// TIA Portal V17 program export: 0 tag tables, 1 data types, 3 data blocks, 1 code blocks (in call order from the OBs), 4 instance data blocks

TYPE "sPut"
// stored: IsFailsafeCompliant false
   STRUCT
      tP : Struct
         REQ : Bool;   // OUT Start sending data
         ERROR : Bool;   // OUT Error sending data
         DONE : Bool;   // OUT sending data completed successfully
         status : Int;
      END_STRUCT;
   END_STRUCT;
END_TYPE

DATA_BLOCK "Data_send_1"   // DB1
{ S7_Optimized_Access := 'FALSE' }
VERSION : 0.1
// stored: AutoNumber true, IsOnlyStoredInLoadMemory false, IsWriteProtectedInAS false
   VAR
      Bool_1 : Bool;
      Bool_2 : Bool;
      Bool_3 : Bool;
      Bool_4 : Bool;
   END_VAR
BEGIN
END_DATA_BLOCK

DATA_BLOCK "dbReceive_PLC1fromPLC2"   // DB7
{ S7_Optimized_Access := 'TRUE' }
VERSION : 0.1
// stored: AutoNumber true, IsOnlyStoredInLoadMemory false, IsWriteProtectedInAS false
   VAR
      Odebrane : Int;
   END_VAR
BEGIN
END_DATA_BLOCK

DATA_BLOCK "dbSend_PLC1toPLC2"   // DB4
{ S7_Optimized_Access := 'TRUE' }
VERSION : 0.1
// stored: AutoNumber true, IsOnlyStoredInLoadMemory false, IsWriteProtectedInAS false
   VAR
      wyslane : Int;
   END_VAR
BEGIN
END_DATA_BLOCK

ORGANIZATION_BLOCK "Main"   // OB1, LAD, ProgramCycle
TITLE = "Main Program Sweep (Cycle)"
{ S7_Optimized_Access := 'TRUE' }
VERSION : 0.1
// stored: AutoNumber true, IsIECCheckEnabled false, SetENOAutomatically false
BEGIN
END_ORGANIZATION_BLOCK

DATA_BLOCK "IEC_Counter_0_DB"   // DB5
{ S7_Optimized_Access := 'TRUE' }
// stored: AutoNumber true, InstanceOfName IEC_COUNTER, OfSystemLibElement IEC_COUNTER, OfSystemLibVersion 1.0
"IEC_COUNTER"
   // VAR RETAIN
   //    CU : Bool;
   //    CD : Bool;
   //    R : Bool;
   //    LD : Bool;
   //    QU : Bool;
   //    QD : Bool;
   //    PV : Int;
   //    CV : Int;
   // END_VAR
BEGIN
END_DATA_BLOCK

DATA_BLOCK "PUT_DB"   // DB2
// stored: AutoNumber true, InstanceOfName PUT_SFB, OfSystemLibElement PUT, OfSystemLibVersion 1.3
"PUT_SFB"
   // VAR_INPUT
   //    REQ : Bool;
   //    ID : Word;
   // END_VAR
   // VAR_OUTPUT
   //    DONE : Bool;
   //    ERROR : Bool;
   //    STATUS : Word;
   // END_VAR
   // VAR_IN_OUT
   //    ADDR_1 : Remote;
   //    ADDR_2 : Remote;
   //    ADDR_3 : Remote;
   //    ADDR_4 : Remote;
   //    SD_1 : Variant;
   //    SD_2 : Variant;
   //    SD_3 : Variant;
   //    SD_4 : Variant;
   // END_VAR
BEGIN
END_DATA_BLOCK

DATA_BLOCK "TRCV_C_DB_1"   // DB6
// stored: AutoNumber true, InstanceOfName TRCV_C, OfSystemLibElement TRCV_C, OfSystemLibVersion 2.1
"TRCV_C"
   // VAR_INPUT
   //    EN_R : Bool;
   //    CONT : Bool;
   //    LEN : UInt;
   // END_VAR
   // VAR_OUTPUT
   //    DONE : Bool;
   //    BUSY : Bool;
   //    ERROR : Bool;
   //    STATUS : Word;
   //    RCVD_LEN : UInt;
   // END_VAR
   // VAR_IN_OUT
   //    CONNECT : TCON_Param;
   //    DATA : Variant;
   //    COM_RST : Bool;
   // END_VAR
   // VAR
   //    sb_FIRSTSTART : Bool;
   //    sb_COMRST : Bool;
   //    sb_CON_EST : Bool;
   //    sb_STARTFB : Bool;
   //    sw_ConID : CONN_OUC;
   //    si_STATE : UInt;
   //    si_JOB : UInt;
   //    s_TCON { S7_SetPoint := 'True'} : TCON;
   //    s_TRCV { S7_SetPoint := 'True'} : TRCV;
   //    s_TDISCON { S7_SetPoint := 'True'} : TDISCON;
   // END_VAR
BEGIN
END_DATA_BLOCK

DATA_BLOCK "TSEND_C_DB"   // DB1
// stored: AutoNumber true, InstanceOfName TSEND_C, OfSystemLibElement TSEND_C, OfSystemLibVersion 2.1
"TSEND_C"
   // VAR_INPUT
   //    REQ : Bool;
   //    CONT : Bool;
   //    LEN : UInt;
   // END_VAR
   // VAR_OUTPUT
   //    DONE : Bool;
   //    BUSY : Bool;
   //    ERROR : Bool;
   //    STATUS : Word;
   // END_VAR
   // VAR_IN_OUT
   //    CONNECT : TCON_Param;
   //    DATA : Variant;
   //    COM_RST : Bool;
   // END_VAR
   // VAR
   //    sb_FIRSTSTART : Bool;
   //    sb_REQ : Bool;
   //    sb_STARTFB : Bool;
   //    sb_CON_EST : Bool;
   //    sb_COMRST : Bool;
   //    si_STATE : UInt;
   //    si_JOB : UInt;
   //    sw_ConID : CONN_OUC;
   //    s_TCON { S7_SetPoint := 'True'} : TCON;
   //    s_TDISCON { S7_SetPoint := 'True'} : TDISCON;
   //    s_TSEND { S7_SetPoint := 'True'} : TSEND;
   // END_VAR
BEGIN
END_DATA_BLOCK
